PROGRAM TESTPRG
VAR
    sequencerTest : Sequencer_Test;
    stepManagerTest : StepManagerBasic_Test;
END_VAR

// Copyright (c) 2024 Loupe (https://loupe.team), provided under the MIT License.

TcUnit.RUN();

END_PROGRAM

(* stored: Version 1.1.0.1
   POU TESTPRG: Id {cb0dada2-790f-48b3-8702-fc17bd7e66f5}, SpecialFunc None *)
